FUNCTION IncUINT : UINT				// Increments the given UINT value
VAR_IN_OUT
	ioNum:	UINT;		// Value to increment
END_VAR

IncUINT := ioNum := ioNum + 1;

END_FUNCTION

(* stored: Version 1.1.0.1, ProductVersion 3.1.4026.18
   POU IncUINT: Id {31d092e6-52cd-4ebf-a77e-eb883b383cb2}, SpecialFunc None *)
